(* CODESYS project FU_bBitPartThrough.xml

Project tree, tasks and I/O mapping:
  function FU_bBitPartThrough [ST]
*)

// FU_bBitPartThrough
//This function changed only the needed bits of a variable
// |**Version**|**Author**| **Date** |**Changes**
// | 1         | NSN      | 16-03-22 | Creation
FUNCTION FU_bBitPartThrough : BYTE
VAR_INPUT
	valueChange		:BYTE;		//Variable to change
	value			:BYTE;		//Value to change bits to
	amount			:BYTE;		//Amount of bits to change
	offset			:BYTE;		//Offset in variable to change bits at
END_VAR

FU_bBitPartThrough		:=		(valueChange AND ROL(GConstants.binaryInvMaskByte[amount],offset)) OR SHL(value AND GConstants.binaryMaskByte[amount],offset);

END_FUNCTION
